Staubli VAL3: onF1Event.pgx

program onF1Event()
  local num l_nValue[4]
  local string l_sItem[4]
  local string l_sMessage
  local num l_nMin[4]
  local num l_nMax[4]
  local bool l_bLarge
  local num l_nKey
begin
  // look if the bButton is enable
  if bButton[0]
    //
    if !bPage
      // normal production page
      if cycleStatus:bCycle==false
        //and cycleStatus:bIsHome==false
        //
        if cycleStatus:nWorkingMode==1
          if isPowered()==false
            call language:message(l_sMessage,201)
            call use:timerDialog(l_sMessage,0)
            do
              l_nKey=getKey()
              if l_nKey==255 or cycleStatus:nWorkingMode!=1
                return
              endIf
              delay(0)
            until isPowered()
          endIf
          l_bLarge=bLarge
          cls()
          cycleStatus:bToHome=true
          wait(cycleStatus:bToHome==false)
          call simulation()
          //
          bLarge=l_bLarge
        else
          call language:message(l_sMessage,92)
          call use:timerDialog(l_sMessage,2)
        endIf
      endIf
    else
      // export the file
      call language:message(l_sMessage,96)
      l_sMessage=l_sMessage+":# actionLog.txt file"
      call use:timerDialog(l_sMessage,0)
      nFile=$fileOpen("actionLog.txt","w")
      $fileSet(nFile,cycleStatus:sLog,size(cycleStatus:sLog))
      $fileClose(nFile)
    endIf
  endIf
end
